(* Schneider Machine Expert - Basic project PLC AI, file version 2.9.0.0 *)
(* ProjectInformations: Name=New project *)

HARDWARE
  Cpu 0: TM221CE16R
  EthernetConfiguration: NetworkName=M221, IpAllocationMode=FixedAddress, IpAddress=192.168.1.50, SubnetMask=255.255.255.0
  SerialLineConfiguration: Baud=Baud19200, Parity=ParityEven, DataBits=DataBits8, StopBits=StopBits1, PhysicalMedium=PhysicalMediumRs485, TransmissionMode=TransmissionModeModbusRtu, SlaveId=1, Addressing=SlaveAddressing
  MastTask: UsePeriodScanMode=false, PeriodScan=100
  FastTask: Period=255
  CpuBehavior: StartingMode=StartAsPreviousState, AutoSaveRamOnEeprom=true, WatchdogPeriod=250

SYMBOLS  (address, symbol, comment, settings)
  %READ_VAR0   [Link(Value(FBComLinkParameterEnums=EthernetLink)), RemoteDeviceId(Value(int=1)), Timeout(Value(int=100)), ObjType(Value(FBComObjTypeParameterEnums=I)), FirstObj(Value(int=0)), Quantity(Value(int=4)), IndexData(Value(int=200))]
  %WRITE_VAR0   [Link(Value(FBComLinkParameterEnums=EthernetLink)), RemoteDeviceId(Value(int=1)), Timeout(Value(int=100)), ObjType(Value(FBComObjTypeParameterEnums=Q)), FirstObj(Value(int=0)), Quantity(Value(int=4)), IndexData(Value(int=100))]

POU New POU
  (* SectionNumber=1 *)

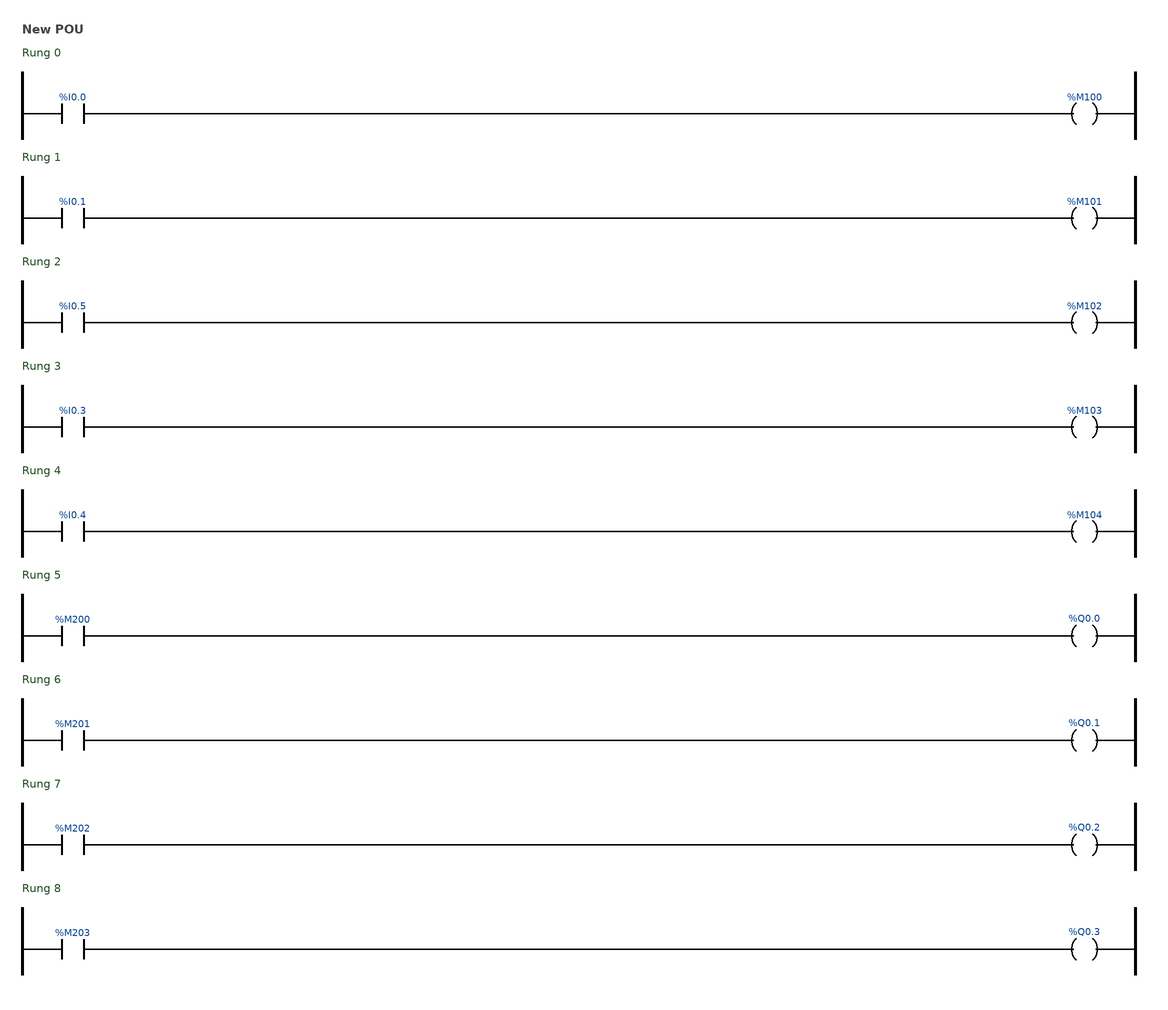

// Rung 0
  LD %I0.0
  ST %M100
  // as ST:
  //   %M100 := %I0.0;

// Rung 1
  LD %I0.1
  ST %M101
  // as ST:
  //   %M101 := %I0.1;

// Rung 2
  LD %I0.5
  ST %M102
  // as ST:
  //   %M102 := %I0.5;

// Rung 3
  LD %I0.3
  ST %M103
  // as ST:
  //   %M103 := %I0.3;

// Rung 4
  LD %I0.4
  ST %M104
  // as ST:
  //   %M104 := %I0.4;

// Rung 5
  LD %M200
  ST %Q0.0
  // as ST:
  //   %Q0.0 := %M200;

// Rung 6
  LD %M201
  ST %Q0.1
  // as ST:
  //   %Q0.1 := %M201;

// Rung 7
  LD %M202
  ST %Q0.2
  // as ST:
  //   %Q0.2 := %M202;

// Rung 8
  LD %M203
  ST %Q0.3
  // as ST:
  //   %Q0.3 := %M203;

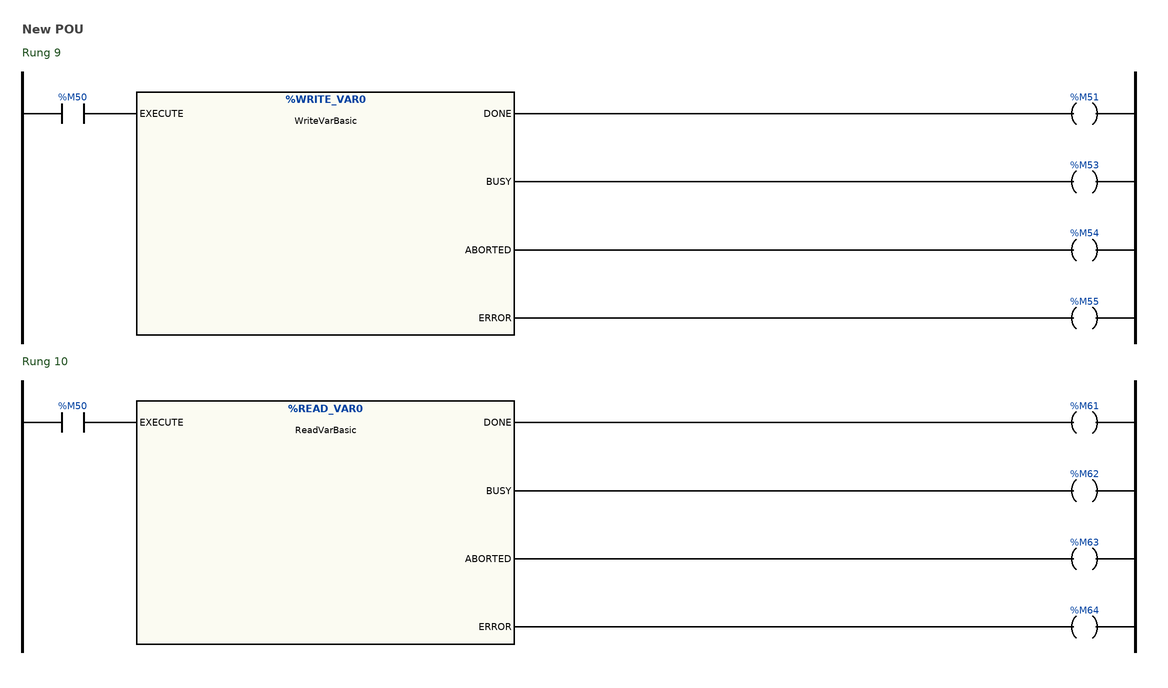

// Rung 9
  BLK %WRITE_VAR0
  LD %M50
  EXECUTE
  OUT_BLK
  LD DONE
  ST %M51
  LD BUSY
  ST %M53
  LD ABORTED
  ST %M54
  LD ERROR
  ST %M55
  END_BLK
  // as ST:
  //   %WRITE_VAR0(EXECUTE := %M50);
  //   %M51 := %WRITE_VAR0.DONE;
  //   %M53 := %WRITE_VAR0.BUSY;
  //   %M54 := %WRITE_VAR0.ABORTED;
  //   %M55 := %WRITE_VAR0.ERROR;

// Rung 10
  BLK %READ_VAR0
  LD %M50
  EXECUTE
  OUT_BLK
  LD DONE
  ST %M61
  LD BUSY
  ST %M62
  LD ABORTED
  ST %M63
  LD ERROR
  ST %M64
  END_BLK
  // as ST:
  //   %READ_VAR0(EXECUTE := %M50);
  //   %M61 := %READ_VAR0.DONE;
  //   %M62 := %READ_VAR0.BUSY;
  //   %M63 := %READ_VAR0.ABORTED;
  //   %M64 := %READ_VAR0.ERROR;
